{attribute 'qualified_only'}
{attribute 'strict'}
TYPE E_ProcessDoor_State :
(
		//GENERIC
	ABORTED				,
	HOMING				,
	READY				,
	MANUAL_MODE			,
	STOPPING			,
	//SPECIFIC FOR EVERY STATION
	OPEN,
	CLOSE,
	DONE				,
	RESET				
);
END_TYPE

(* stored: Version 1.1.0.1, ProductVersion 3.1.4026.18
   DUT E_ProcessDoor_State: Id {4099e79a-dd09-4eee-a9ea-147d9a547a32} *)
